(* Passes one DWORD read across the arbiter bridge. The caller links the raw PDO value and derives
   bridge health elsewhere (e.g. FB_SubSysToArbiter_IO.bBridgeOk) and passes both in each cycle; this
   FB owns no hardware links. Integers have no invalid-bit-pattern to sanitize, so it holds the last
   trusted value while the bridge is down. Error carries only the test override; fault on bad comms
   via the bridge FB's bBridgeConfirmedBad in the caller. *)
FUNCTION_BLOCK FB_FallibleDwordFromEtherCAT
IMPLEMENTS I_FallibleDword
VAR_INPUT
    i_bBridgeOk : BOOL;
    i_nValue : DWORD;
END_VAR
VAR_OUTPUT
    {attribute 'pytmc' := '
        pv: Value
        io: i
    '}
    nValue : DWORD;
END_VAR
VAR
    nLastValidValue : DWORD;
    bOverride : BOOL;
    bOverrideError : BOOL;
    nOverrideValue : DWORD;
END_VAR


IF i_bBridgeOk THEN
    nLastValidValue := i_nValue;
END_IF

nValue := SEL(bOverride, SEL(i_bBridgeOk, nLastValidValue, i_nValue), nOverrideValue);


PROPERTY Error : BOOL
GET

Error := SEL(bOverride, FALSE, bOverrideError);
END_GET
END_PROPERTY


PROPERTY Value : DWORD
GET

Value := THIS^.nValue;
END_GET
END_PROPERTY

END_FUNCTION_BLOCK

(* stored: Version 1.1.0.1
   POU FB_FallibleDwordFromEtherCAT: Id {a1b2c3d4-0102-4001-8001-000000000201}, SpecialFunc None
   Property Error: Id {a1b2c3d4-0102-4001-8001-000000000202}
   Get Get: Id {a1b2c3d4-0102-4001-8001-000000000203}
   Property Value: Id {a1b2c3d4-0102-4001-8001-000000000204}
   Get Get: Id {a1b2c3d4-0102-4001-8001-000000000205} *)
